Staubli VAL3: onF1Event.pgx

program onF1Event()
  local string l_sPalletName
  local num i
begin
  // look if the bButton is enable
  if bButton[0]
    call pallet:reset()
  endIf
end
